// TIA Portal V19 export
TYPE "Analogic_SensorManagement_Data"
// stored: Access Published
   STRUCT
      OffsetValue : LReal;
      OffsetValid : Bool;
   END_STRUCT;
END_TYPE
